// TwinCAT 3 PLC project PLC
// ProgramVersion: 3.1.4024.0
// libraries:
//   Tc2_Standard, * (Beckhoff Automation GmbH)
//   Tc2_System, * (Beckhoff Automation GmbH)
//   Tc3_Module, * (Beckhoff Automation GmbH)
// project tree:
//   / PlcTask.TcTTO
//   POUs/ MAIN.TcPOU, POU_FBD.TcPOU, SrT.TcPOU

CONFIGURATION PLC
    RESOURCE PLC ON TwinCAT3
        TASK PlcTask(INTERVAL := T#10ms, PRIORITY := 20);
        PROGRAM MAIN WITH PlcTask : MAIN;
    END_RESOURCE
END_CONFIGURATION

// ---- POUs/MAIN.TcPOU
PROGRAM MAIN
VAR
	// Q1
	//loop : INT := 1;
	
	// Q2
	//tempurature : REAL := 26.5;
	
	// Q3
	// INT : num1 := 1;	
	// Type and name are wrong way round
	// Should be:
	// num1 : INT := 1;
	
	// Q4
	// num1 := 1;	
	// No variable type
	// Should be:
	// num1 : INT := 1;
	
	// Q5
	// Refer to "SrT"
	
	// Q6
	// C will be TRUE
	
	// Q7
	// C will be TRUE
	
	// Q8
	// 
	
END_VAR

POU_FBD();

END_PROGRAM

// ---- POUs/POU_FBD.TcPOU
PROGRAM POU_FBD
VAR
	input : BOOL;
	output : BOOL := false;
END_VAR

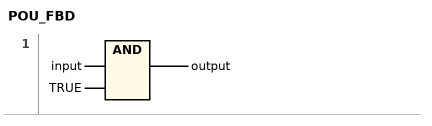
// NETWORK 1
output := input AND TRUE;

END_PROGRAM

// ---- POUs/SrT.TcPOU
PROGRAM POU_ST
VAR
	num1 : INT := 1;
 	num2 : INT := 2;
 	res : INT := 0;
	
	op1 : INT := 0;
	op2 : INT := 0;
END_VAR

// res will be -5
// 1 / 2 -> 0.5 -> 0
// 0 - 5 -> -5

op1 := num1;
op2 := num2;
res := op1 / op2 - 5;

END_PROGRAM
